Staubli VAL3: remGetESTOP.pgx

program remGetESTOP(string& sReturn[] (dimensions=1))
  local string sEstop
begin
  // Return the ESTOP status
  //
  logMsg("call remGetESTOP")
  switch esStatus()
    case 0
      sEstop="INACTIVE"
    break
    case 1
      sEstop="STOPPED"
    break
    case 2
      sEstop="READY"
    break
  endSwitch
  sReturn="GETESTOP "+sEstop
end
